// TIA Portal V20 export
DATA_BLOCK "za_TraceCodeGeneration_DB"   // DB263
// stored: InstanceOfName za_TraceCodeGeneration, InstanceOfType FB
"za_TraceCodeGeneration"
   // VAR_INPUT
   //    ComponentType : String;
   //    MfgSiteId : String;
   //    Shift : String;
   //    LineIdentifier : String;
   //    GMPartNumber : String;
   //    SignalForTC_Creation : Bool;
   //    SignalForSN_Increment : Bool;
   //    SignalForSN_Reset : Bool;
   //    SignalForTCBuffer_Clear : Bool;
   //    AlwaysON : Bool;
   //    ProgramID : String;
   //    System_Clock_1s_Pulse : Bool;
   // END_VAR
   // VAR_OUTPUT
   //    TracebilityCode : String;
   //    TracebilityCode_Ready : Bool;
   //    Tracecode : Array[1..20] of Char;
   //    PartNumber : Array[1..8] of Char;
   // END_VAR
   // VAR
   //    TCtimer : TON_TIME;
   // END_VAR
   // VAR RETAIN
   //    instCounter : CTU_DINT;
   //    statPrevTraceBilityCode : String;
   // END_VAR
   // VAR
   //    statPrevDailySequenceNumber : DInt;
   //    TraceCodeData { ExternalAccessible := 'False'; ExternalVisible := 'False'; ExternalWritable := 'False'} : Array[0..20] of String[26];
   //    TraceCellNumber { ExternalAccessible := 'False'; ExternalVisible := 'False'; ExternalWritable := 'False'} : Array[0..20] of USInt;
   //    statTracecodeBuffer : Array[1..20] of Char;
   //    statPartNumberBuffer : Array[1..8] of Char;
   //    statTracecodeBufferCnt : UInt;
   //    statPartNumberBufferCnt : UInt;
   // END_VAR
BEGIN
END_DATA_BLOCK
